# EPICS autosave request: andorApp/Db/andorCCD_settings.req
$(P)$(R)AndorCooler
$(P)$(R)AndorAccumulatePeriod
$(P)$(R)AndorShutterMode
$(P)$(R)AndorShutterExTTL
$(P)$(R)PALFilePath
$(P)$(R)AndorPreAmpGain
$(P)$(R)AndorEMGain
$(P)$(R)AndorEMGainMode
$(P)$(R)AndorEMGainAdvanced
$(P)$(R)AndorADCSpeed
$(P)$(R)AndorReadOutMode
file "ADBase_settings.req", P=$(P), R=$(R)
file "NDFile_settings.req", P=$(P), R=$(R)
